{attribute 'hide_all_locals'}
FUNCTION_BLOCK Mc2Halt EXTENDS TaskBase
VAR_INPUT
END_VAR
VAR_OUTPUT
END_VAR
VAR
	mcHalt : Tc2_MC2.MC_Halt;
	_axis : REFERENCE TO Tc2_MC2.AXIS_REF;
	_Halt : BOOL;
END_VAR

METHOD Abort : BOOL
mchalt.Execute := FALSE;
_busy := FALSE;
_Halt := FALSE;
Abort := TRUE;
State := 0;
END_METHOD

METHOD Cycle : BOOL
VAR_INPUT
END_VAR
CASE State OF
	0:
		IF _Halt THEN
			_done := FALSE;
			_error := FALSE;
			_busy := TRUE;
			mcHalt.Execute := TRUE;
			IF mcHalt.Busy THEN
				State := 10;
				_Halt := FALSE;
			END_IF
		END_IF
	
	10:
		IF NOT mcHalt.Busy THEN
			IF mcHalt.Done THEN
				_done := TRUE;
			ELSIF mcHalt.Error THEN
				_error := TRUE;
			END_IF
			_busy := FALSE;
			mcHalt.Execute := FALSE;
			State := 0;
		END_IF
END_CASE

mcHalt(Axis := _axis);
END_METHOD

METHOD Execute : BOOL
VAR_INPUT
END_VAR
Execute := _Halt := true;
END_METHOD

METHOD FB_init : BOOL
VAR_INPUT
	bInitRetains : BOOL; // if TRUE, the retain variables are initialized (warm start / cold start)
	bInCopyCode : BOOL;  // if TRUE, the instance afterwards gets moved into the copy code (online change)
	axis : reference TO AXIS_REF;
END_VAR
_axis REF= axis;
END_METHOD

END_FUNCTION_BLOCK

(* stored: Version 1.1.0.1, ProductVersion 3.1.4024.12
   POU Mc2Halt: Id {a1da82b8-b5e2-423a-81ce-89f8e220d6ba}, SpecialFunc None
   Method Abort: Id {f78f1251-51d0-4d67-9a04-2fb8762c04c1}
   Method Cycle: Id {de80207a-320b-426e-a8d0-0a658b69f5c9}
   Method Execute: Id {ac08f8cb-3ea1-46cb-8397-98b2e5ffacc4}
   Method FB_init: Id {54531f04-5f04-4e0e-b4c4-371c5398b9d6} *)
